// TIA Portal V20 export
DATA_BLOCK "AxisConfigBackUp_DB"   // DB176
// stored: MemoryReserve 100
   VAR
      ManualSave : Bool;
   END_VAR
   VAR RETAIN
      DR1 : Struct
         cmJROutPnPLeftPositionX : Array[0..15] of "LBC_typeAxis64PosSetPosition";
      END_STRUCT;
      DR2 : Struct
         cmJROutPnPLeftPositionZ : Array[0..15] of "LBC_typeAxis64PosSetPosition";
      END_STRUCT;
      DR3 : Struct
         cmJROutPnPRightPositionX : Array[0..15] of "LBC_typeAxis64PosSetPosition";
      END_STRUCT;
      DR4 : Struct
         cmJROutPnPRightPositionZ : Array[0..15] of "LBC_typeAxis64PosSetPosition";
      END_STRUCT;
      DR5 : Struct
         cmTopTapingX : Array[0..15] of "LBC_typeAxis64PosSetPosition";
      END_STRUCT;
      DR6 : Struct
         cmTopTapingY : Array[0..15] of "LBC_typeAxis64PosSetPosition";
      END_STRUCT;
      DR7 : Struct
         cmJrFixStageX : Array[0..15] of "LBC_typeAxis64PosSetPosition";
      END_STRUCT;
      DR8 : Struct
         cmJrFixStageC : Array[0..15] of "LBC_typeAxis64PosSetPosition";
      END_STRUCT;
      DR9 : Struct
         cmSideTapingX : Array[0..15] of "LBC_typeAxis64PosSetPosition";
      END_STRUCT;
      DR10 : Struct
         cmSideTapingY : Array[0..15] of "LBC_typeAxis64PosSetPosition";
      END_STRUCT;
      DR11 : Struct
         cmHipotThicknessZ : Array[0..15] of "LBC_typeAxis64PosSetPosition";
      END_STRUCT;
      DR12 : Struct
         cmTransferPPLeftX : Array[0..15] of "LBC_typeAxis64PosSetPosition";
      END_STRUCT;
      DR13 : Struct
         cmTransferPPLeftY : Array[0..15] of "LBC_typeAxis64PosSetPosition";
      END_STRUCT;
      DR14 : Struct
         cmTransferPPLeftZ : Array[0..15] of "LBC_typeAxis64PosSetPosition";
      END_STRUCT;
      DR15 : Struct
         cmTransferPPRightX : Array[0..15] of "LBC_typeAxis64PosSetPosition";
      END_STRUCT;
      DR16 : Struct
         cmTransferPPRightY : Array[0..15] of "LBC_typeAxis64PosSetPosition";
      END_STRUCT;
      DR17 : Struct
         cmTransferPPRightZ : Array[0..15] of "LBC_typeAxis64PosSetPosition";
      END_STRUCT;
      DR18 : Struct
         cmJrUnloadingX : Array[0..15] of "LBC_typeAxis64PosSetPosition";
      END_STRUCT;
      DR19 : Struct
         cmJrUnloadingZ : Array[0..15] of "LBC_typeAxis64PosSetPosition";
      END_STRUCT;
      DR20 : Struct
         cmJrUnloadingC : Array[0..15] of "LBC_typeAxis64PosSetPosition";
      END_STRUCT;
   END_VAR
BEGIN
END_DATA_BLOCK
